FUNCTION_BLOCK Path EXTENDS Spline
VAR_INPUT
	xWPL: 	ARRAY [0..100] OF LREAL; // raw x data
	yWPL: 	ARRAY [0..100] OF LREAL; // raw y data
	radius: LREAL;
END_VAR
VAR
	x: 					ARRAY [0..100] OF LREAL; // preprocessed x data
	y: 					ARRAY [0..100] OF LREAL; // preprocessed x data
	transitions: 		ARRAY [0..99] OF LREAL;
	subsplines: 		ARRAY [0..99] OF Spline;
	nmbOfSubsplines, nmbOfPreprocessedWaypoints:	INT;
	i, j, k: INT;
	
	xTmpBezier,yTmpBezier:    		ARRAY [0..2] OF LREAL;
 	xTmpLinear,yTmpLinear:    		ARRAY [0..1] OF LREAL;
	start, end:						RobotPoseSimple;
END_VAR

preprocessWaypointlist();

nmbOfSubsplines := 2*nmbOfPreprocessedWaypoints-3;

FOR i := 1 TO nmbOfSubsplines BY 2 DO
	k := 0;
	//extract relevant points for bezier curve creation
	FOR j := (3*i-1)/2 TO (3*i-1)/2+2 BY 1 DO
		xTmpBezier[k] := x[j]; 
		yTmpBezier[k] := y[j];
		k := k + 1;
	END_FOR  
	subsplines[i]:= BezierCurve(x:=xTmpBezier, y:=yTmpBezier, radius:=radius);
END_FOR

//last Segment is always linear
xTmpLinear[0] := x[0];
xTmpLinear[1] := x[1];
yTmpLinear[0] := y[0];
yTmpLinear[1] := y[1];
subsplines[0] := LinearSpline(x := xTmpLinear, y := yTmpLinear);

//last Segment is always linear
xTmpLinear[0] := x[nmbOfPreprocessedWaypoints-2];
xTmpLinear[1] := x[nmbOfPreprocessedWaypoints-1];
yTmpLinear[0] := y[nmbOfPreprocessedWaypoints-2];
yTmpLinear[1] := y[nmbOfPreprocessedWaypoints-1];
subsplines[nmbOfSubsplines-1] := LinearSpline(x := xTmpLinear, y := yTmpLinear);

//generate the linear segments in between
FOR i := 2 TO nmbOfSubsplines-2 BY 2 DO
	//extract relevant waypoints
	end		  		:= subsplines[i+1].startPointVal; //end is the start point of the next segment
	start  		  := subsplines[i-1].endPointVal;	  //start is the endpoint of the prev segment
	xTmpLinear[0] := start.x;
	xTmpLinear[1] := end.x;
	yTmpLinear[0] := start.y;
	yTmpLinear[1] := end.y;
	subsplines[i] := LinearSpline(x:=xTmpLinear, y:= yTmpLinear);
END_FOR

calculateLength();
calculateTransitions();

startPoint := subsplines[0].startPointVal;
endPoint   := subsplines[nmbOfSubsplines-1].endPointVal;

METHOD PROTECTED  calculateLength : LREAL
VAR_INPUT
END_VAR
VAR
	i: INT;
END_VAR
calculateLength := 0;
FOR i := 0 TO nmbOfSubsplines-1 DO
	calculateLength := calculateLength + subsplines[i].length;
END_FOR
END_METHOD

METHOD calculateTransitions
VAR_INPUT
END_VAR
VAR
	i : INT;
END_VAR
transitions[0] := 0;
FOR i := 0 TO nmbOfSubsplines-2 DO
	transitions[i+1] := transitions[i] + subsplines[i].length;
END_FOR
END_METHOD

METHOD  diff : RobotPoseSimple
VAR_INPUT
	arcLength: LREAL;
	order: INT := 1;
END_VAR
VAR
	subspline: 				Spline;
	arcOffset, deltaTheta: 	LREAL;
	dPos: RobotPoseSimple;
	
END_VAR
getSubsplineToPoint(arcLength := arcLength,
					subspline => subspline,
					arcOffset => arcOffset);
deltaTheta:= endPoint.theta - startPoint.theta; 		
dPos 		:= subspline.diff(arcLength := arcOffset, order:= order);	
diff.x 		:= dPos.x;
diff.y 		:= dPos.y;	
CASE order OF
	1:
		diff.theta  := deltaTheta*pi/(2*lengthVar)*SIN(pi/lengthVar*arcLength);
	2:
		diff.theta 	:= deltaTheta*EXPT(pi,2)/(2*EXPT(lengthVar,2))*SIN(pi/lengthVar*arcLength);
ELSE
		diff.x      := -1;
		diff.y 		:= -1;
END_CASE
END_METHOD

METHOD getDiscontinuousSwitchtingPointCandidate : ARRAY  [0..99] OF LREAL
VAR_INPUT
END_VAR
VAR
	i : INT := 0;
END_VAR
FOR i := 1 TO nmbOfSubsplines-2 DO
	getDiscontinuousSwitchtingPointCandidate[i-1]  := transitions[i];
END_FOR
END_METHOD

METHOD PUBLIC  getPoint : RobotPoseSimple
VAR_INPUT
	arcLength: LREAL;
END_VAR
VAR
	subspline: Spline;
	arcOffset: LREAL;
END_VAR
getSubsplineToPoint(arcLength := arcLength,
					subspline => subspline,
					arcOffset => arcOffset);
getPoint := subspline.getPoint(arcLength:= arcOffset);
END_METHOD

METHOD getSubsplineToPoint : Spline
VAR_INPUT
	arcLength: LREAL;
END_VAR

VAR_OUTPUT
	subspline: Spline;
	arcOffset: LREAL;
END_VAR
arcOffset := arcLength;
FOR i := 0 TO nmbOfSubsplines-1 DO
	IF arcOffset -subsplines[i].length < 0 THEN
		subspline := subsplines[i];
		EXIT;
	ELSE
		arcOffset := arcOffset -subsplines[i].length;
	END_IF
END_FOR
END_METHOD

PROPERTY length : LREAL
GET
END_GET
SET
END_SET
END_PROPERTY

METHOD preprocessWaypointlist 
VAR_IN_OUT
END_VAR
VAR 
	i : 				INT 			:= 0;
	nextIDX: 			INT;
	phi1, phi2: 		LREAL;
END_VAR

x[0] := xWPL[0];
y[0] := yWPL[0];
nextIDX := 1;

FOR i := 1 TO 99 DO
	//exit if last point is reached, last valid point is last point in preprocessed list
	IF xWPL[i+1] = -1 AND yWPL[i+1] = -1 THEN
		x[nextIDX] := xWPL[i];	
		y[nextIDX] := yWPL[i];
		EXIT;
	END_IF	

	phi1 := ATAN2(yWPL[i]-yWPL[i-1],xWPL[i]-xWPL[i-1]);
	phi2 := ATAN2(yWPL[i+1]-yWPL[i],xWPL[i+1]-xWPL[i]);
	IF phi1 <> phi2 THEN
		x[nextIDX] := xWPL[i];	
		y[nextIDX] := yWPL[i];
		nextIDX := nextIDX +1;
	END_IF
END_FOR
nmbOfPreprocessedWaypoints := nextIDX +1;
END_METHOD

END_FUNCTION_BLOCK

(* stored: Version 1.1.0.1, ProductVersion 3.1.4024.11
   POU Path: Id {95fe6ec8-af15-4fc0-b4c5-550c7aba9b73}, SpecialFunc None
   Method calculateLength: Id {fa9150c3-1548-4fad-bc03-2a7bdbb95fff}
   Method calculateTransitions: Id {52dbb64c-0f38-4919-8d0f-8a50326cf34d}
   Method diff: Id {c435850d-099e-4883-9ebf-b0187bee6499}
   Method getDiscontinuousSwitchtingPointCandidate: Id {cfaa726c-df69-48c1-84c4-a6f3a80b3d25}
   Method getPoint: Id {edc81ff7-b7ad-4aac-a526-a3258fc65de9}
   Method getSubsplineToPoint: Id {d9693a58-8dc8-4612-b85b-8d181f60b2f3}
   Property length: Id {9758eca7-15ca-47fd-ba8e-a9ee5447051a}
   Get Get: Id {e0813d43-db58-4b26-90b5-a965f7cab4d5}
   Set Set: Id {229f1c6f-dee2-45a0-af40-ce116e09667f}
   Method preprocessWaypointlist: Id {eb2abc10-4b35-4a8b-a276-447cab2534b7} *)
